TYPE ST_BigBagPar :
STRUCT
    rBagTargetMass_SP       : REAL;
    rBagFullToleranceKg     : REAL;
END_STRUCT
END_TYPE

(* stored: Version 1.1.0.1, ProductVersion 3.1.4024.16
   DUT ST_BigBagPar: Id {2e081202-c3d3-43dc-a61c-40a3157de105} *)
